Universal Robots PolyScope program: 5-movec.urp

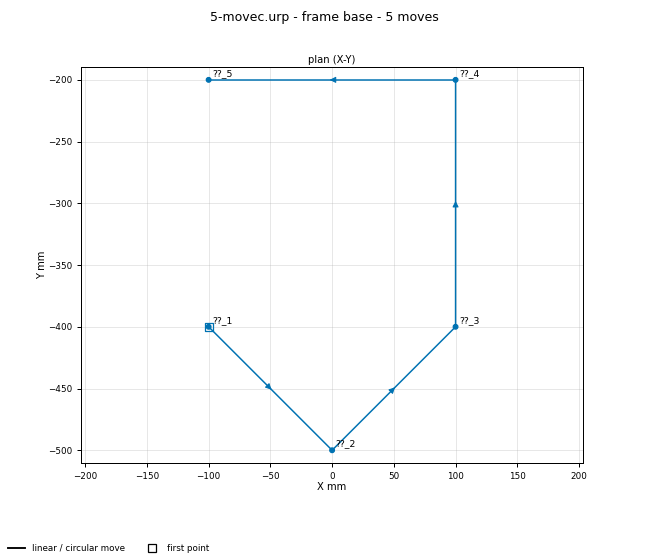
[picture p0: tool path of 5-movec.urp in frame base, 5 of 5 moves have a stored position in this frame; points joined in program order, loops and branches not executed]
ProgramRoot directory=/home/ur/ursim-3.1/programs/basic training/5-movec; kinematics=(a=[0, -0.425, -0.39225, 0, 0, 0], d=[0.08916, 0, 0, 0.10915, 0.09465, 0.0823], alpha=[1.5708, 0, 0, 1.5708, -1.5708, 0], deltaTheta=[0, 0, 0, 0, 0, 0], status=notInitialized); lastSavedInVersion=(project__name=Polyscope, major__version=3, minor__version=1, svn__revision=17195, build__date=Mar 11 2015, 13:02:28); name=5-movec; programVersion=(project__name=Polyscope, major__version=3, minor__version=1, svn__revision=17195, build__date=Mar 11 2015, 13:02:28); robotEnvironmentFileName=default; serialNumberRobot=2014350001
  MainProgram cartesianAcceleration=1.2; cartesianSpeed=0.25; jointAcceleration=1.3962634015954636; jointSpeed=1.0471975511965976; sharedProcessMoveBlendRadius=0.025; motionType=JOINT_SPACE
    Move cartesianAcceleration=1.2; cartesianSpeed=0.25; jointAcceleration=1.3962634015954636; jointSpeed=1.0471975511965976; sharedProcessMoveBlendRadius=0.025; motionType=PROCESS_MOVE
      Waypoint blendRadius=0.05; cartesianAcceleration=1.2; cartesianSpeed=0.25; jointAcceleration=1.3962634015954636; jointSpeed=1.0471975511965976; nextMotionTime=2.0; stoppoint=true; useSharedBlendParameter=true; useSharedParameters=true; outputFlangePose=(pos=(x=-0.10000000065989616, y=-0.40000000104212996, z=0.1999999982306596), rot=(x=-0.0012209830283997337, y=3.116276481240887, z=0.0388919161681283)); position=TCP in base x=-100 y=-400 z=200 mm, rx=-0.0012 ry=3.1163 rz=0.0389 rad; joints [-88.988, -88.3, -127.491, -55.614, 91.461, 0.95] deg; positionType=FIXED_POSITION; waypointPoseInFeatureCoordinates=(pos=(x=-0.09999996819589951, y=-0.40000005265404437, z=0.1999999632555712), rot=(x=-0.0012210995530369398, y=3.1162764787073427, z=0.0388923209577584)); name=路点_1
      CircleMove description=Circle_Move_description; name=CircleMove
        Waypoint blendRadius=0.05; cartesianAcceleration=1.2; cartesianSpeed=0.25; jointAcceleration=1.3962634015954636; jointSpeed=1.0471975511965976; nextMotionTime=2.0; stoppoint=true; useSharedBlendParameter=true; useSharedParameters=true; outputFlangePose=(pos=(x=-1.6712002807148182E-10, y=-0.4999999994986338, z=0.19999998792029502), rot=(x=-0.0012208534573162541, y=3.1162765026745682, z=0.03889211050910082)); position=TCP in base x=0 y=-500 z=200 mm, rx=-0.0012 ry=3.1163 rz=0.0389 rad; joints [-77.679, -99.924, -114.856, -56.312, 91.708, 12.26] deg; positionType=FIXED_POSITION; waypointPoseInFeatureCoordinates=(pos=(x=9.653020530813008E-8, y=-0.49999997873435936, z=0.20000009704921962), rot=(x=-0.0012211638662894828, y=3.116276433100459, z=0.03889172047786868)); name=路点_2
        Waypoint blendRadius=0.0; cartesianAcceleration=1.2; cartesianSpeed=0.25; jointAcceleration=1.3962634015954636; jointSpeed=1.0471975511965976; nextMotionTime=2.0; useSharedBlendParameter=true; useSharedParameters=true; outputFlangePose=(pos=(x=0.09999999967038797, y=-0.399999999670377, z=0.1999999879202973), rot=(x=-0.001220853457340838, y=3.116276502674616, z=0.038892110508861634)); position=TCP in base x=100 y=-400 z=200 mm, rx=-0.0012 ry=3.1163 rz=0.0389 rad; joints [-61.016, -88.295, -127.75, -54.511, 91.949, 28.93] deg; positionType=FIXED_POSITION; waypointPoseInFeatureCoordinates=(pos=(x=0.09999990769115596, y=-0.3999999728939928, z=0.1999998399702372), rot=(x=-0.0012205781234201267, y=3.11627671400097, z=0.03889276118000279)); name=路点_3
      Waypoint blendRadius=0.05; cartesianAcceleration=1.2; cartesianSpeed=0.25; jointAcceleration=1.3962634015954636; jointSpeed=1.0471975511965976; nextMotionTime=2.0; stoppoint=true; useSharedBlendParameter=true; useSharedParameters=true; outputFlangePose=(pos=(x=0.10000003093008784, y=-0.19999997720808027, z=0.2000000202491838), rot=(x=-0.0012209058669235583, y=3.116276536037026, z=0.038892034429442064)); position=TCP in base x=100 y=-200 z=200 mm, rx=-0.0012 ry=3.1163 rz=0.0389 rad; joints [-35.055, -51.443, -149.443, -68.76, 91.996, 54.906] deg; positionType=FIXED_POSITION; waypointPoseInFeatureCoordinates=(pos=(x=0.10000003093004557, y=-0.19999997679952106, z=0.20000002024915683), rot=(x=-0.0012209058668588384, y=3.1162765360370175, z=0.03889203442947606)); name=路点_4
      Waypoint blendRadius=0.05; cartesianAcceleration=1.2; cartesianSpeed=0.25; jointAcceleration=1.3962634015954636; jointSpeed=1.0471975511965976; nextMotionTime=2.0; stoppoint=true; useSharedBlendParameter=true; useSharedParameters=true; outputFlangePose=(pos=(x=-0.10000000034079462, y=-0.19999999965923698, z=0.1999998396364955), rot=(x=-0.001221229174446227, y=3.1162768257265276, z=0.038892683103097445)); position=TCP in base x=-100 y=-200 z=200 mm, rx=-0.0012 ry=3.1163 rz=0.0389 rad; joints [-87.972, -51.697, -148.925, -70.758, 91.486, 1.966] deg; positionType=FIXED_POSITION; waypointPoseInFeatureCoordinates=(pos=(x=-0.10000003279081764, y=-0.19999996476675833, z=0.19999978392221096), rot=(x=-0.001221002579610083, y=3.11627687011649, z=0.03889320766147045)); name=路点_5
